// Brief: Setup Arm Init
FUNCTION_BLOCK PUBLIC FB_SetupCtrlHold EXTENDS FB_SetupArmCtrlBase
VAR_INPUT
END_VAR
VAR_OUTPUT
END_VAR
VAR
	m_initState :INT :=0;
END_VAR

END_FUNCTION_BLOCK

(* stored: Version 1.1.0.1, ProductVersion 3.1.4024.12
   POU FB_SetupCtrlHold: Id {acc6ed82-034a-420c-8162-3225c33c4b38}, SpecialFunc None *)
